INTERFACE I_Station_LinkedList

METHOD AddHeadValue : ST_STATION_LIST_RESULT
VAR_INPUT
  stData        : ST_STATION_MOVER_DATA;
END_VAR
END_METHOD

METHOD AddTailValue : ST_STATION_LIST_RESULT
VAR_INPUT
  stData          : ST_STATION_MOVER_DATA;
END_VAR
END_METHOD

PROPERTY Count : UDINT
GET
END_GET
END_PROPERTY

PROPERTY Data : ARRAY[1..MAX_LIST_NODES] OF ST_STATION_MOVER_DATA
GET
END_GET
END_PROPERTY

PROPERTY Free : UDINT
GET
END_GET
END_PROPERTY

METHOD GetHead : ST_STATION_LIST_RESULT
VAR_INPUT
END_VAR
END_METHOD

METHOD InitList : BOOL
END_METHOD

PROPERTY Nodes : ARRAY[0..MAX_LIST_NODES] OF T_LinkedListEntry
GET
END_GET
END_PROPERTY

METHOD RemoveHeadValue : ST_STATION_LIST_RESULT
VAR_INPUT
END_VAR
END_METHOD

END_INTERFACE

(* stored: Version 1.1.0.1
   Itf I_Station_LinkedList: Id {dd484fce-224b-419a-af89-8e194e6f0f8f}
   Method AddHeadValue: Id {491b864b-0410-4bb2-92de-05086038ca3d}
   Method AddTailValue: Id {4c4254ea-f88a-40ad-a9f4-62474bc9576f}
   Property Count: Id {13585bb8-5d8c-4682-b8f6-224f0eae4137}
   Get Get: Id {0d2bfead-4fc3-43eb-9405-11e1fb232717}
   Property Data: Id {d9b9eccf-96f4-49d8-8bb6-8e390555534a}
   Get Get: Id {b5f5a393-d2c3-4638-bbbe-96360278b669}
   Property Free: Id {0636d0f8-e6c3-4156-aabb-a406711b494a}
   Get Get: Id {da36bfb3-d42d-4a1e-8697-6464409ab178}
   Method GetHead: Id {80557974-c328-46d3-ad7d-f79ea3efe37a}
   Method InitList: Id {d571c6f7-bb47-41b1-a4e9-90c9f58a1f31}
   Property Nodes: Id {746a3164-3f40-4d67-98c2-384edaefe4d6}
   Get Get: Id {2778367f-60b9-4097-a3d6-28a169036571}
   Method RemoveHeadValue: Id {d1dc343b-9b1d-4c58-829f-10c7517e6a07} *)
